PROGRAM PRG_Compilation
VAR
END_VAR

END_PROGRAM

(* stored: Version 1.1.0.1, ProductVersion 3.1.4024.15
   POU PRG_Compilation: Id {4756b3be-b3eb-4597-bf5d-6355bd41fd4b}, SpecialFunc None *)
